(* CODESYS project My first FB.project

Project tree, tasks and I/O mapping:
  Device : CODESYS Control Win V3, 3S - Smart Software Solutions GmbH, version 3.5.15.30
    application Application
      libraries: Standard, * (System)
      task MainTask (cyclic, interval t#20ms, priority 1) calls PLC_PRG_FBD
      program PLC_PRG_ST [ST]
      function block SumAndSub [ST]
      program PLC_PRG_FBD [FBD]
*)

// Device/Application/PLC_PRG_FBD
PROGRAM PLC_PRG_FBD
VAR
	SumAndSub_0: SumAndSub;
	
	X : REAL := 20;
	Y : REAL := 3;
	
	R_Sum : REAL;
	R_Sub : REAL;
	
END_VAR

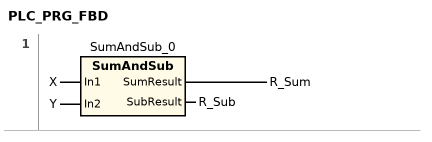
// NETWORK 1
SumAndSub_0(In1 := X, In2 := Y, SubResult => R_Sub); // SumAndSub
R_Sum := SumAndSub_0.SumResult;

END_PROGRAM

// Device/Application/SumAndSub
FUNCTION_BLOCK SumAndSub
VAR_INPUT
	In1 : REAL;
	In2 : REAL;
END_VAR
VAR_OUTPUT
	SumResult : REAL;
	SubResult : REAL;
END_VAR
VAR
END_VAR

SumResult := In1 + In2;
SubResult := In1 - In2;

END_FUNCTION_BLOCK

// Device/Application/PLC_PRG_ST
PROGRAM PLC_PRG_ST
VAR
	A : REAL := 11;
	B : REAL := 5;
	Somma : REAL;
	Sottrazione : REAL;
	MyFB : SumAndSub;
END_VAR

MyFB(In1 := A, In2 := B);

Somma := MyFB.SumResult;
Sottrazione := MyFB.SubResult;

END_PROGRAM
